// TIA Portal V16 export
// export: Created 2022-01-12T14:34:27.0342547Z, ExportSetting WithDefaults, DisplayName Totally Integrated Automation Portal, DisplayVersion V16 Update 4, DisplayName TIA Portal Version Control Interface, DisplayVersion V16 Update 2, DisplayName TIA Portal Openness, DisplayVersion V16 Update 4, DisplayName STEP 7 Professional, DisplayVersion V16 Update 4, DisplayName STEP 7 Safety, DisplayVersion V16, DisplayName WinCC Professional, DisplayVersion V16 Update 4
TYPE "typProgram"
// stored: IsFailsafeCompliant false
   STRUCT
      nazwaFunkcji : Int;
      nazwaKroku : Int;
      numerKroku : Int;
      numerKrMycia : Int;
      zadana1 : Real;
      aktualna1 : Real;
      zadana2 : Real;
      aktualna2 : Real;
      opóżnienie : Real;
   END_STRUCT;
END_TYPE
